{attribute 'qualified_only'}
{attribute 'strict'}
TYPE E_SDSHomingState :
(
    INIT := 0,
    WAIT_NOT_BUSY,
    TRIGGER_HOMING,
    WAIT_FOR_HOMED,
    HOMED
) UINT;
END_TYPE

(* stored: Version 1.1.0.1
   DUT E_SDSHomingState: Id {e1dfb655-f154-005d-003b-eb56c249e79f} *)
